PROGRAM SpeedControl_SIM
VAR
	
//Boolean values for determining the speed at which the motors are running in a controlled and called fashion.
	bEncCallMade1   	: BOOL := FALSE;
	bEncCallMade2   	: BOOL := FALSE;
	bEncCallMade3   	: BOOL := FALSE;
	bEncCallMade4   	: BOOL := FALSE;
	bMotor1Running  	: BOOL := GVL_VAR.bMotor1Running;
	bMotor2Running  	: BOOL := GVL_VAR.bMotor2Running;
	bMotor3Running  	: BOOL := GVL_VAR.bMotor3Running;
	bMotor4Running  	: BOOL := GVL_VAR.bMotor4Running;
	bProgramStarted 	: BOOL := GVL_VAR.bStartButton;
	bMotorsHaveStarted  : BOOL := GVL_VAR.bMotorsHaveStarted;
	bFirstReading		: BOOL;
	bSpeedCheck1Pass	: BOOL;
	bSpeedCheck2Pass	: BOOL;
	bSpeedCheck3Pass	: BOOL;
	bSpeedCheck4Pass	: BOOL;
	
//Global Variables into which the encoder values will be stored.
	iEncoder1Val 		: INT := GVL_VAR.diMotorEncoder1;
	iEncoder2Val 		: INT := GVL_VAR.diMotorEncoder2;
	iEncoder3Val 		: INT := GVL_VAR.diMotorEncoder3;
	iEncoder4Val 		: INT := GVL_VAR.diMotorEncoder4;
	iEncoderPPR			: INT := GVL_VAR.iEncoderPPR;
	
//Hysteresis of the encoders...
	iEncoder1Hys 		: INT := GVL_VAR.diEncoder1Hysteresis;
	iEncoder2Hys 		: INT := GVL_VAR.diEncoder2Hysteresis;
	iEncoder3Hys 		: INT := GVL_VAR.diEncoder3Hysteresis;
	iEncoder4Hys 		: INT := GVL_VAR.diEncoder4Hysteresis;
	
//Retrieve the speed settings for the scope of the flow and assign them to local variable names...
	iGlobalSpeedSetting : INT := GVL_VAR.iSetGlobalSpeed;
	iMotor1Speed 		: INT := GVL_VAR.iMotor1GlobalSpeed;
	iMotor2Speed 		: INT := GVL_VAR.iMotor2GlobalSpeed;
	iMotor3Speed 		: INT := GVL_VAR.iMotor3GlobalSpeed;
	iMotor4Speed 		: INT := GVL_VAR.iMotor4GlobalSpeed;
	
//This is primarily used for storing the encoder values and comparisons between motor speeds...
	iMotor1SpeedA		: INT := 0;
	iMotor2SpeedA		: INT := 0;
	iMotor3SpeedA		: INT := 0;
	iMotor4SpeedA		: INT := 0;
	
//Timer functions for controlling the encoder value polling
	tEncCallMadeTimer 	: TON;
	timerDone 			: BOOL := FALSE;
END_VAR

(*Simulated Program*)
//This is for determining the speed of the motors and displaying it on the UI. It is also
// responsible for making sure that all of the motors are indeed running the same speed through measurement.
//This measurement is then taken and it adjusts the speed of the motors accordingly (just for the sake of testing the logic of course)
//If after a certain amount of adjustments the speed still seems unbalanced, THEN the machine will switch off the motor controls and flag a product JAM.
//Give the command to start the motors

IF bProgramStarted THEN
	GVL_VAR.bStartMotor1 := TRUE;
	GVL_VAR.bStartMotor2 := TRUE;
	GVL_VAR.bStartMotor3 := TRUE;
	GVL_VAR.bStartMotor4 := TRUE;
ELSE 
	GVL_VAR.bStartMotor1 := FALSE;
	GVL_VAR.bStartMotor2 := FALSE;
	GVL_VAR.bStartMotor3 := FALSE;
	GVL_VAR.bStartMotor4 := FALSE;
END_IF

//Confirm whether or not the motors have started...
IF bMotor1Running AND bMotor2Running AND bMotor3Running AND bMotor4Running THEN
	//Set the global variable GVL_VAR.bMotorsHaveStarted to TRUE if ALL of the run feedback signals are TRUE
	GVL_VAR.bMotorsHaveStarted := TRUE;
ELSE
	//Set the global variable GVL_VAR.bMotorsHaveStarted to FALSE if NOT ALL of the run feedback signals are TRUE
	GVL_VAR.bMotorsHaveStarted := FALSE;
END_IF

WHILE bMotorsHaveStarted DO 
	//Start the timer for orderky data calls
	IF NOT timerDone THEN
		tEncCallMadeTimer(IN := TRUE, PT:=T#100MS, Q=> timerDone);
	
		IF NOT bEncCallMade1 AND tEncCallMadeTimer.ET = T#25MS  THEN
			iMotor1Speed := iEncoder1Val - iEncoder1Hys;
			iMotor1SpeedA := iEncoder1Val;
			//ensure that the process isn't executed every single new scan cycle by using a boolean trigger
			bEncCallMade1 := TRUE;
			//now the iMotor1Speed Can be formatted and made available to the UI
		END_IF
		
		IF NOT bEncCallMade2 AND tEncCallMadeTimer.ET = T#50MS  THEN
			iMotor2Speed := iEncoder2Val - iEncoder3Hys;
			iMotor2SpeedA := iEncoder2Val;
			//ensure that the process isn't executed every single new scan cycle by using a boolean trigger
			bEncCallMade2 := TRUE;
			//now the iMotor2Speed Can be formatted and made available to the UI
		END_IF
	
		IF NOT bEncCallMade3 AND tEncCallMadeTimer.ET = T#75MS  THEN
			iMotor3Speed := iEncoder3Val - iEncoder3Hys;
			iMotor3SpeedA := iEncoder3Val;
			//ensure that the process isn't executed every single new scan cycle by using a boolean trigger
			bEncCallMade3 := TRUE;
			//now the iMotor3Speed Can be formatted and made available to the UI
		END_IF
	
		IF NOT bEncCallMade4 AND tEncCallMadeTimer.ET = T#100MS  THEN
			iMotor4Speed := iEncoder4Val - iEncoder4Hys;
			iMotor4SpeedA := iEncoder4Val;
			//ensure that the process isn't executed every single new scan cycle by using a boolean trigger
			bEncCallMade4 := TRUE;
			//now the iMotor4Speed Can be formatted and made available to the UI
		END_IF

		IF timerDone AND bEncCallMade4 THEN
			bEncCallMade1 := FALSE;
			bEncCallMade2 := FALSE;
			bEncCallMade3 := FALSE;
			bEncCallMade4 := FALSE;
			tEncCallMadeTimer.IN := FALSE;
			tEncCallMadeTimer.Q := FALSE;
			bFirstReading := TRUE;
			
		END_IF
	END_IF


	
END_WHILE
//Reference in essense a PID controller for all of these motors
//Compare all of the motor's speeds with the main speed setting
WHILE bFirstReading DO
	
	IF iMotor1Speed = iGlobalSpeedSetting THEN
		bSpeedCheck1Pass := TRUE;
		GVL_VAR.bIncreaseSpeed1 := FALSE;
		GVL_VAR.bDecreaseSpeed1 := FALSE;
	ELSE IF iMotor1Speed > iGlobalSpeedSetting THEN
			//DECREASE motor speed!
			bSpeedCheck1Pass := FALSE;
			GVL_VAR.bDecreaseSpeed1 := TRUE;
			
		ELSE //INCREASE motor speed!
			bSpeedCheck1Pass := FALSE;
			GVL_VAR.bIncreaseSpeed1 := TRUE;
		END_IF
	END_IF
	
	IF iMotor2Speed = iGlobalSpeedSetting THEN
		bSpeedCheck2Pass := TRUE;
		GVL_VAR.bIncreaseSpeed2 := FALSE;
		GVL_VAR.bDecreaseSpeed2 := FALSE;

	ELSE IF iMotor2Speed > iGlobalSpeedSetting THEN
		//DECREASE motor speed!
		bSpeedCheck2Pass := FALSE;
		GVL_VAR.bDecreaseSpeed2 := TRUE;
		
		ELSE //INCREASE motor speed!
			bSpeedCheck2Pass := FALSE;
			GVL_VAR.bIncreaseSpeed2 := TRUE;
		END_IF
	END_IF
	
	IF iMotor3Speed = iGlobalSpeedSetting THEN
		bSpeedCheck3Pass := TRUE;
		GVL_VAR.bIncreaseSpeed3 := FALSE;
		GVL_VAR.bDecreaseSpeed3 := FALSE;
	
	ELSE IF iMotor3Speed > iGlobalSpeedSetting THEN
		//DECREASE motor speed!
		bSpeedCheck3Pass := FALSE;
		GVL_VAR.bDecreaseSpeed3 := TRUE;
		
		ELSE //INCREASE motor speed!
			bSpeedCheck3Pass := FALSE;
			GVL_VAR.bIncreaseSpeed3 := TRUE;
		END_IF
	
	END_IF
	
	
	IF iMotor4Speed = iGlobalSpeedSetting THEN
		bSpeedCheck4Pass := TRUE;
		GVL_VAR.bIncreaseSpeed4 := FALSE;
		GVL_VAR.bDecreaseSpeed4 := FALSE;
		
	ELSE IF iMotor4Speed > iGlobalSpeedSetting THEN
		//DECREASE motor speed!
		bSpeedCheck4Pass := FALSE;
		GVL_VAR.bDecreaseSpeed4 := TRUE;
		
		ELSE //INCREASE motor speed!
			bSpeedCheck4Pass := FALSE;
			GVL_VAR.bIncreaseSpeed4 := TRUE;
		END_IF
	
	END_IF

	
END_WHILE

END_PROGRAM

(* stored: Version 1.1.0.1, ProductVersion 3.1.4024.12
   POU SpeedControl_SIM: Id {0a562722-591e-4057-8289-46035a92b04b}, SpecialFunc None *)
